PROGRAM Axis04_Status
VAR
//System_Bit
	Always_ON	:	BOOL	:=TRUE	;//상시 ON 
	Always_OFF	:	BOOL	:=FALSE	;//상시 OFF
	
//Motor_Command
	Axis04_Status_01: MC_ReadStatus;
	Axis04_Position_Read_01: MC_ReadActualPosition;
	Axis04_Velocity_Read_01: MC_ReadActualVelocity;
	Axis04_Reset_01: MC_Reset;
	Axis04_Stop_01: MC_Stop;
	Torque_Down : UINT := 1500;
	Torque_Up : UINT := 1500;
END_VAR
VAR // added by the converter: edge detectors and wires of the graphical bodies
    _rt1 : R_TRIG;
END_VAR

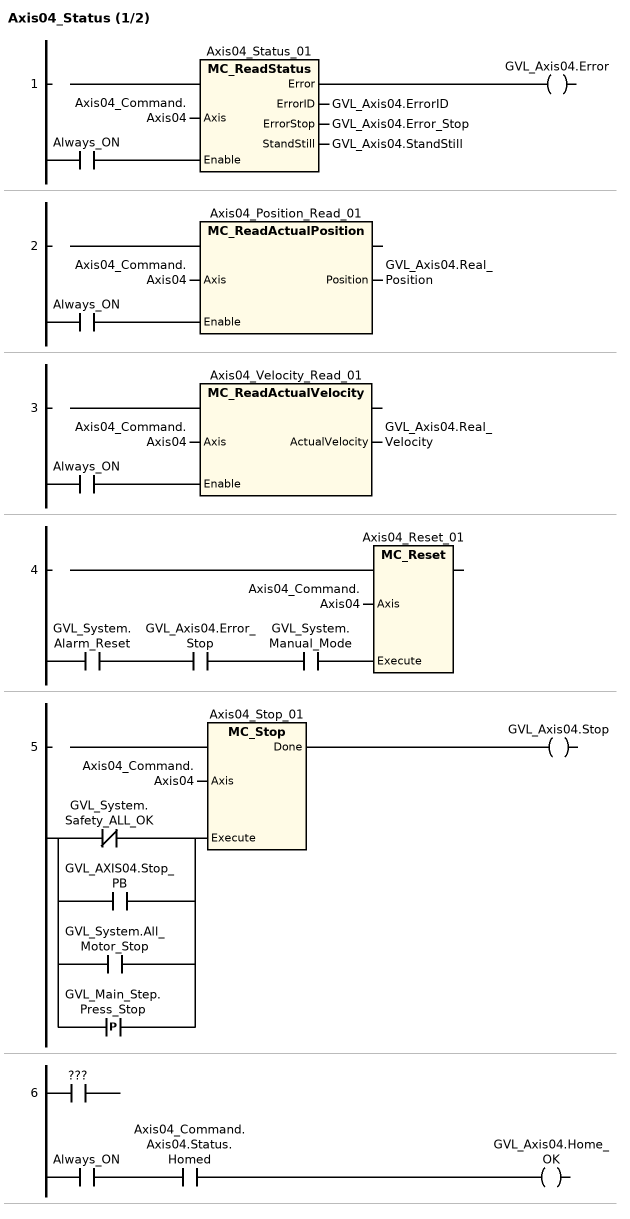
// NETWORK 1
Axis04_Status_01(
    Axis := Axis04_Command.Axis04,
    Enable := Always_ON,
    Error => GVL_Axis04.Error,
    ErrorID => GVL_Axis04.ErrorID,
    ErrorStop => GVL_Axis04.Error_Stop,
    StandStill => GVL_Axis04.StandStill); // MC_ReadStatus

// NETWORK 2
Axis04_Position_Read_01(
    Axis := Axis04_Command.Axis04,
    Enable := Always_ON,
    Position => GVL_Axis04.Real_Position); // MC_ReadActualPosition

// NETWORK 3
Axis04_Velocity_Read_01(
    Axis := Axis04_Command.Axis04,
    Enable := Always_ON,
    ActualVelocity => GVL_Axis04.Real_Velocity); // MC_ReadActualVelocity

// NETWORK 4
Axis04_Reset_01(Axis := Axis04_Command.Axis04, Execute := GVL_System.Alarm_Reset AND GVL_Axis04.Error_Stop AND GVL_System.Manual_Mode); // MC_Reset

// NETWORK 5
_rt1(CLK := GVL_Main_Step.Press_Stop);
Axis04_Stop_01(Axis := Axis04_Command.Axis04, Execute := NOT GVL_System.Safety_ALL_OK OR GVL_AXIS04.Stop_PB OR GVL_System.All_Motor_Stop OR _rt1.Q); // MC_Stop
GVL_Axis04.Stop := Axis04_Stop_01.Done;

// NETWORK 6
GVL_Axis04.Home_OK := Always_ON AND Axis04_Command.Axis04.Status.Homed;

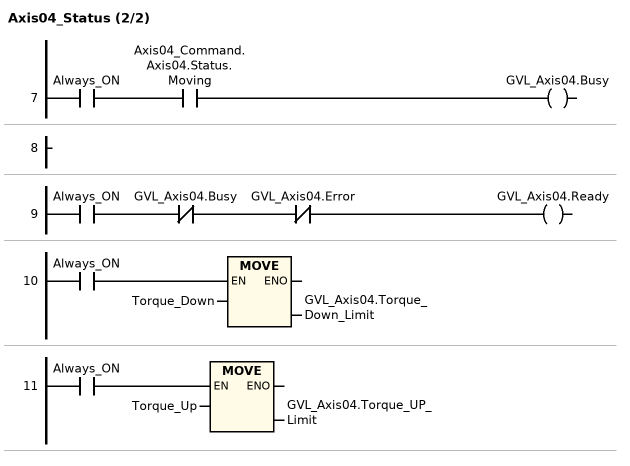
// NETWORK 7
GVL_Axis04.Busy := Always_ON AND Axis04_Command.Axis04.Status.Moving;

// NETWORK 8

// NETWORK 9
GVL_Axis04.Ready := Always_ON AND NOT GVL_Axis04.Busy AND NOT GVL_Axis04.Error;

// NETWORK 10
IF Always_ON THEN GVL_Axis04.Torque_Down_Limit := Torque_Down; END_IF

// NETWORK 11
IF Always_ON THEN GVL_Axis04.Torque_UP_Limit := Torque_Up; END_IF

END_PROGRAM

(* stored: Version 1.1.0.1, ProductVersion 3.1.4024.16
   POU Axis04_Status: Id {1f8022e4-871d-472b-a064-e15cacdef46d}, SpecialFunc None *)
